INTERFACE IWaitBlock

END_INTERFACE

(* stored: Version 1.1.0.1, ProductVersion 3.1.4024.6
   Itf IWaitBlock: Id {3f105005-e8ee-4b29-ba29-506e6ca5be5b} *)
